INTERFACE I_GigeRegister EXTENDS I_CH_Object

{attribute 'monitoring' := 'call'}
PROPERTY AllReadDone : BOOL
GET
END_GET
SET
END_SET
END_PROPERTY

{attribute 'monitoring' := 'call'}
PROPERTY AllWriteDone : Bool
GET
END_GET
SET
END_SET
END_PROPERTY

//Rewrite parameters if necessary, e.g. after a connection interruption
METHOD RewriteParameters : HRESULT
VAR_INPUT
END_VAR
END_METHOD

END_INTERFACE

(* stored: Version 1.1.0.1, ProductVersion 3.1.4024.15
   Itf I_GigeRegister: Id {13381513-d2a4-43fb-a7f9-ac173fc14f06}
   Property AllReadDone: Id {3a6158c4-5a5b-437c-8363-ea2d9270c4bb}
   Get Get: Id {811dab00-6e17-445b-a49f-3eaa60deb4e2}
   Set Set: Id {b0c2be25-0e5c-4b36-9a56-94eaa8df3ba8}
   Property AllWriteDone: Id {13dd2b53-7af7-402e-898a-7c60b6866d76}
   Get Get: Id {b1b7b5c5-944d-4b72-b665-3b2af42e129f}
   Set Set: Id {45b58d8c-606c-4c98-9163-360c2c0e1a99}
   Method RewriteParameters: Id {c802142d-eea6-4a9a-9345-dce314cd96c3} *)
